// TIA Portal V20 export
ORGANIZATION_BLOCK "CyclicInterrupt"   // OB30, SCL, CyclicInterrupt
{ S7_Optimized_Access := 'TRUE' }
// stored: SetENOAutomatically false
   VAR_INPUT
      Initial_Call : Bool;   // Initial call of this OB
      Event_Count : Int;   // Events discarded
   END_VAR
BEGIN
   REGION Description head
       //==================================================================================
       // POSALUX Swiss SA / (C) Copyright 2026
       //----------------------------------------------------------------------------------
       // Title: Hardware interrupt
       // Comment/Function: OB30
       // Author: Fabien WALDT
       // Engineering: TIA Portal v20
       //----------------------------------------------------------------------------------
       // Change log table:
       // Version  | Date     | Expert in charge | Changes applied
       //----------------------------------------------------------------------------------
       // 00.00.01 | 20260501 | WFA              | First released version
       //==================================================================================
   END_REGION

   REGION Machine temperature cooling PID
       "CONT_C_Clim_DB"(COM_RST := "DB_Temperature".sPIDRestart,
                        MAN_ON := FALSE,
                        P_SEL := TRUE,
                        I_SEL := TRUE,
                        INT_HOLD := "DB_Temperature".sPIDHoldI,
                        D_SEL := TRUE,
                        CYCLE := T#1s,
                        SP_INT := "DB_HMISetting".TemperatureCoolingSetpoint,
                        PV_IN := "DB_AnalogInputs".sClimTemperature.sSWRealValue,
                        GAIN := "DB_Temperature".sP,
                        TI := "DB_Temperature".sI,
                        TD := "DB_Temperature".sD,
                        DEADB_W := 0.1,
                        LMN_HLM := 100,
                        LMN_LLM := 0,
                        LMN => "DB_AnalogOutputs".sPropValveClimSetPoint.sSWRealValue);
   END_REGION
END_ORGANIZATION_BLOCK
